{attribute addProperty BoxType "AT2050-0500-0020"}
{attribute addProperty Id "A_0093_AT2020_5250_0019_AT2020_5250AT2020_3DCFC8D064080"}
{attribute addProperty CRC "2290062503"}
{attribute addProperty SizeInBites "640"}
{attribute addProperty SizeInBytes "80"}
TYPE A_0051_AT2050_0500_0020_887F94A7 EXTENDS AT2050_9506A482 :
STRUCT
	{attribute addProperty Name "A_0093_AT2020_5250_0019_AT2020_5250"}
	A_0093_AT2020_5250_0019_AT2020_5250 : AT2020_3DCFC8D0;
END_STRUCT
END_TYPE

(* stored: Version 1.2.0.0, ProductVersion 3.1.4024.9
   DUT A_0051_AT2050_0500_0020_887F94A7: Id {c149f856-c0b1-4cb4-8156-52bcd43452ff} *)
